TYPE ST_CM_SERVO_STS :
STRUCT
	done: BOOL;
	outPos: BOOL;
	nearPos: BOOL;
	homed: BOOL;
	power: BOOL;
	error: BOOL;
	errorCode: UDINT;
	pos: REAL;
END_STRUCT
END_TYPE

(* stored: Version 1.1.0.1, ProductVersion 3.1.4024.12
   DUT ST_CM_SERVO_STS: Id {6a4841bb-341f-45cf-8ef2-9e574f651f1e} *)
